{attribute 'qualified_only'}
VAR_GLOBAL
fbPLCDBRead    	: FB_PLCDBReadEvt (sNetID := '', tTimeout := T#5S);
fbPLCDBWrite    :  FB_PLCDBWriteEvt(sNetID := '', tTimeout := T#5S);
END_VAR

(* stored: Version 1.1.0.1, ProductVersion 3.1.4024.9
   GVL GVL: Id {bde25adf-eec3-434c-8133-e5b7a9baf7eb} *)
